FUNCTION_BLOCK PULSE (* Composite Function Block Type *)
  (* Standard: 61499-2 *)
  (* Version 0.0, 5/25/2016, Andrei, nxtControl GmbH, template *)
  PACKAGE Main;
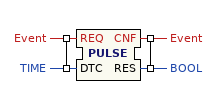
  EVENT_INPUT
    REQ WITH DTC; (* Normal Execution Request *)
  END_EVENT
  EVENT_OUTPUT
    CNF WITH RES; (* Execution Confirmation *)
  END_EVENT
  VAR_INPUT
    DTC : TIME; (* Input event qualifier *)
  END_VAR
  VAR_OUTPUT
    RES : BOOL; (* Output event qualifier *)
  END_VAR
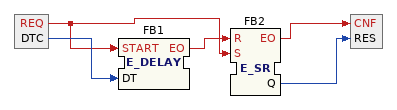
  FBS
    FB1 : E_DELAY;
    FB2 : E_SR;
  END_FBS
  EVENT_CONNECTIONS
    FB1.EO TO FB2.R;
    REQ TO FB1.START;
    REQ TO FB2.S;
    FB2.EO TO CNF;
  END_CONNECTIONS
  DATA_CONNECTIONS
    DTC TO FB1.DT;
    FB2.Q TO RES;
  END_CONNECTIONS
END_FUNCTION_BLOCK
